FUNCTION F_ToAnyType : ST_AnyType
VAR_INPUT
	anyArg	: ANY;
END_VAR

F_ToAnyType.pValue := anyArg.pValue;
F_ToAnyType.nSize := anyArg.diSize;
F_ToAnyType.TypeClass := anyArg.TypeClass;

END_FUNCTION

(* stored: Version 1.1.0.1, ProductVersion 3.1.4024.12
   POU F_ToAnyType: Id {42ad9bab-d5a0-49d5-a1f7-133ba38a0dc8}, SpecialFunc None *)
